// Mitsubishi GX Works2 project: 2stepper   PLC: FX2N/FX2NC

PROGRAM MAIN
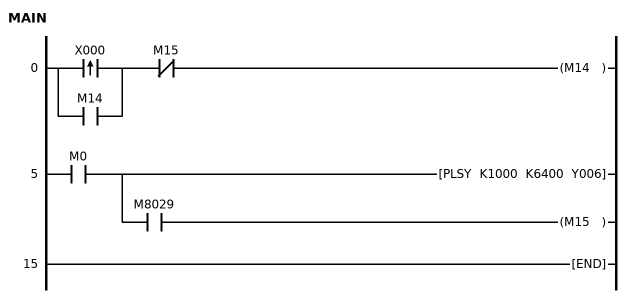
0     LDP     X000
      OR      M14
      ANI     M15
      OUT     M14
5     LD      M0
      PLSY    K1000 K6400 Y006
      AND     M8029
      OUT     M15
15    END
END_PROGRAM
